FUNCTION F_ET2Sec : REAL
VAR_INPUT
	IN: TIME;
	SecScale: REAL;
END_VAR
VAR
	r1: REAL;
END_VAR


r1:= TIME_TO_REAL(IN);
IF r1 > 0 THEN
	F_ET2Sec := r1 / SecScale;
ELSE
	F_ET2Sec := 0;	
END_IF

END_FUNCTION

(* stored: Version 1.1.0.1, ProductVersion 3.1.4024.12
   POU F_ET2Sec: Id {e1839d72-0a7d-4d4d-bfd6-33337bb05106}, SpecialFunc None *)
